# EPICS substitutions: mc09/tpmacApp/Db/motor.substitutions
file "db/motor.db"
{
pattern
{P,              M,                     MOTOR,  PORT,  ADDR,  DESC,  DTYP,      MRES,   EGU,  PREC,  ALIAS }
{"XF:16IDC-OP",  "{CRL-Ax:Z}Mtr",       "M0",   "P0",  1,     "Z",   asynMotor, "3.125E-3",  "mm", 2,     ""    }
{"XF:16IDC-OP",  "{CRL-Ax:Z1}Mtr",      "M0",   "P0",  2,     "Z1",  asynMotor, "3.125E-3",  "mm", 2,     ""    }
{"XF:16IDC-ES",  "{Stg:WAXS1-Ax:X}Mtr", "M0",   "P0",  3,     "X",   asynMotor, "7.938E-4",  "mm", 2,     ""    }
{"XF:16IDC-ES",  "{Stg:WAXS1-Ax:Z}Mtr", "M0",   "P0",  4,     "Z",   asynMotor, "1.563E-4",  "mm", 2,     ""    }
{"XF:16IDC-ES",  "{Stg:WAXS1-Ax:Y}Mtr", "M0",   "P0",  5,     "Y",   asynMotor, "7.938E-4",  "mm", 2,     ""    }
{"XF:16IDC-ES",  "{Stg:WAXS2-Ax:X}Mtr", "M0",   "P0",  6,     "X",   asynMotor, "7.938E-4",  "mm", 2,     ""    }
{"XF:16IDC-ES",  "{Stg:WAXS2-Ax:Z}Mtr", "M0",   "P0",  7,     "Z",   asynMotor, "1.563E-4",  "mm", 2,     ""    }
{"XF:16IDC-ES",  "{Stg:WAXS2-Ax:Y}Mtr", "M0",   "P0",  8,     "Y",   asynMotor, "7.938E-4",  "mm", 2,     ""    }
}
